PROGRAM MAIN
VAR
	stop: BOOL;
	start: BOOL;
	R1: BOOL;
	R2: BOOL;
	weight: INT;
	binASorter: BOOL;
	binBSorter: BOOL;
END_VAR

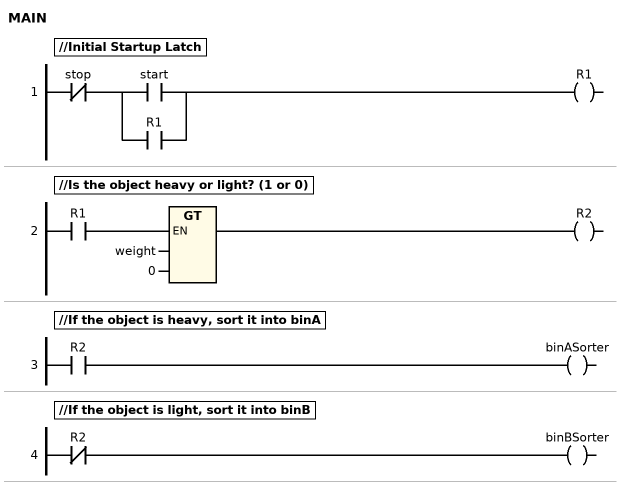
// NETWORK 1
// label: //Initial Startup Latch
R1 := NOT stop AND (start OR R1);

// NETWORK 2
// label: //Is the object heavy or light? (1 or 0)
R2 := R1 AND weight > 0;

// NETWORK 3
// label: //If the object is heavy, sort it into binA
binASorter := R2;

// NETWORK 4
// label: //If the object is light, sort it into binB
binBSorter := NOT R2;

END_PROGRAM

(* stored: Version 1.1.0.1, ProductVersion 3.1.4024.12
   POU MAIN: Id {e02ea011-b87b-45a9-84e2-2f3b89ca1890}, SpecialFunc None *)
